ABB RobotStudio station: Projekt.rspag

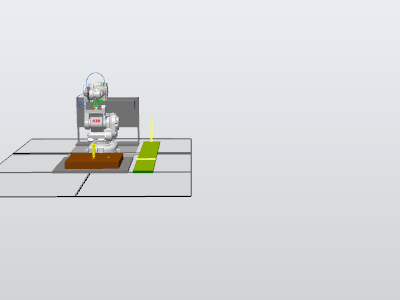
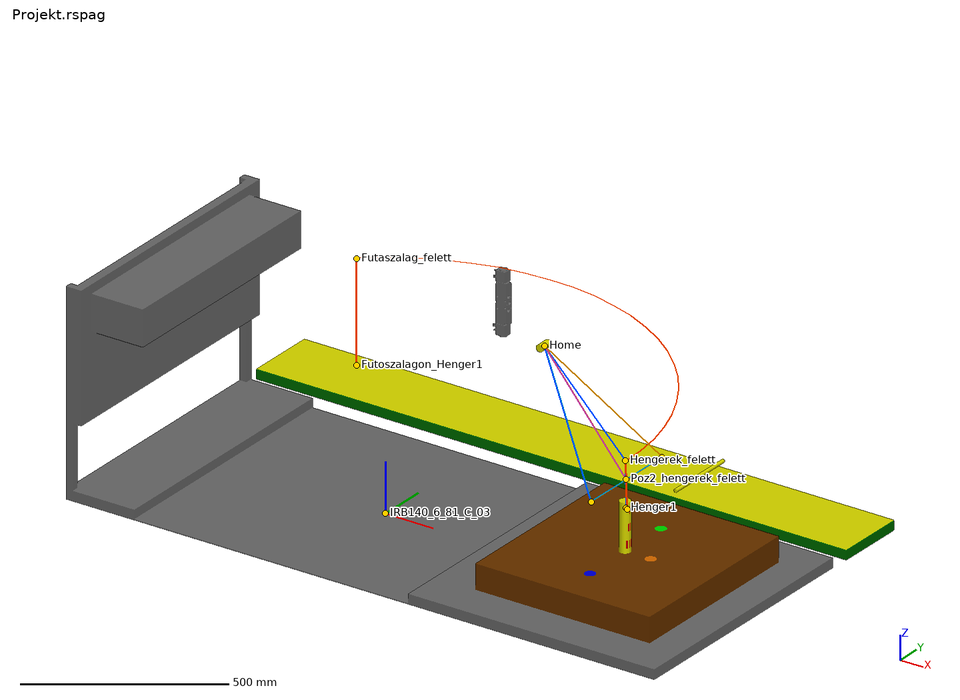
[picture v1: parts stored in the station drawn from their meshes, with robot base, taught points and paths (robot models come from the ABB library and are not in the file)]
--- station ---
Station hanoi_2022_RW6 (saved by RobotStudio 25.1.11167.1)
Controller IRB140_6_81
  mechanical unit ROB_1: IRB140_6_81_C_03, 6 joints, base frame (0, 0, 0) mm
Layout (positions relative to the parent item):
  - Henger1 [part] at (700, 0, 186) mm, rotated rx 0 ry 0 rz 180 deg, size 30.5 x 29.9 x 45 mm
  - Poz1 [part] at (700, 150, 96) mm, size 30 x 29.8 x 0 mm
  - Poz3 [part] at (700, 0, 96) mm, size 30 x 29.8 x 0 mm
  - SmatMefogo [smart component] at (450, 0, 647) mm, rotated rx -180 ry 0 rz -179.16 deg
      signals: DI Megfog, DI Elenged
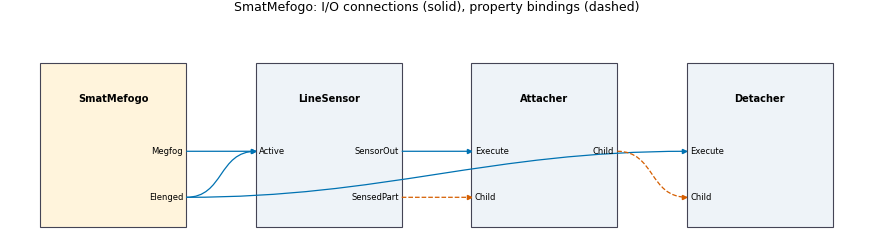
      connections:
        SmatMefogo.Megfog -> LineSensor.Active
        LineSensor.SensorOut -> Attacher.Execute
        SmatMefogo.Elenged -> LineSensor.Active
        SmatMefogo.Elenged -> Detacher.Execute
        LineSensor.SensedPart => Attacher.Child
        Attacher.Child => Detacher.Child
    - Megfogo [mechanism, from Libraries\Megfogo.rslib] at (0, 0, 0) mm, rotated rx 0 ry 0 rz -90 deg; joint values [0] (rad or m)
    - MegfogoTool [mechanism] at (0, 0, 0) mm
        TCP MyNewTool at (-15, 0, 70) mm, rotated rx -90 ry 0 rz -90 deg
        links: Dummy
    - LineSensor [smart component, from Components\LineSensor.rslib]
        properties: Start=[-0.0125 0.018 0.07]; End=[-0.0125 -0.019 0.07]; Radius=0.01; SensedPart=Henger1; SensedPoint=[0.704940063476562 -0.133748397827148 0.231000228881836]; Length=0.037; Tag=(none); SenseMultiple=false
      - _sensorPart_ [part], size 20 x 37 x 20 mm
    - Attacher [smart component, from Components\Attacher.rslib]
        properties: Parent=Megfogo; Flange=0; Child=Henger1; Mount=false; Offset=[0 0 0]; Orientation=[0 0 0]
    - Detacher [smart component, from Components\Detacher.rslib]
        properties: Child=Henger1; KeepPosition=true
  - SmartFSzalag [smart component] at (24.45, 0, 0) mm
      signals: DI Activate, DO SzalagErzekel
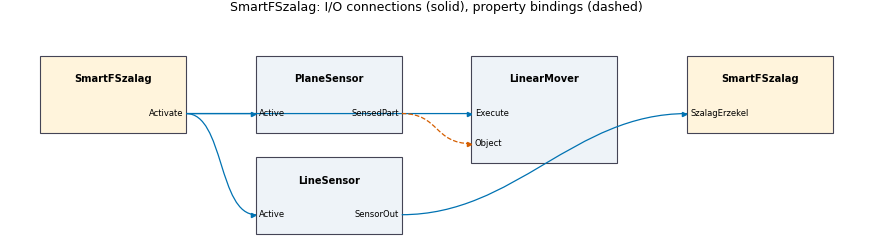
      connections:
        SmartFSzalag.Activate -> LinearMover.Execute
        SmartFSzalag.Activate -> PlaneSensor.Active
        SmartFSzalag.Activate -> LineSensor.Active
        LineSensor.SensorOut -> SmartFSzalag.SzalagErzekel
        PlaneSensor.SensedPart => LinearMover.Object
    - LinearMover [smart component, from Components\LinearMover.rslib]
        properties: Object=(none); Direction=[1 0 0]; Speed=0.1; Reference=Global; ReferenceObject=(none)
    - PlaneSensor [smart component, from Components\PlaneSensor.rslib]
        properties: Origin=[-0.7 0.425 0.027]; Axis1=[1.725 0 0]; Axis2=[0 0.2 0]; SensedPart=(none); Tag=(none); SenseMultiple=false
      - _sensorPart_ [part], size 1725 x 200 x 0 mm
    - FutoSzalag [part] at (-700, 425, 0) mm, size 1725 x 200 x 25 mm
    - LineSensor [smart component, from Components\LineSensor.rslib]
        properties: Start=[0.525 0.625 0.045]; End=[0.525 0.425 0.045]; Radius=0.005; SensedPart=(none); SensedPoint=[0 0 0]; Length=0.2; Tag=(none); SenseMultiple=false
      - _sensorPart_ [part], size 10 x 200 x 10 mm
  - Poz2 [part] at (-100, -100, 71) mm, size 30 x 29.8 x 0 mm
  - Asztal [part], size 1720 x 745 x 567 mm
  - Henger2 [part] at (700, 0, 141) mm, rotated rx 0 ry 0 rz 180 deg, size 30.5 x 29.9 x 45 mm
  - Henger3 [part] at (700, 0, 96) mm, rotated rx 0 ry 0 rz 180 deg, size 30.5 x 29.9 x 45 mm
  - Doboz [part] at (444.29, -260.35, 25.4) mm, size 510 x 540 x 70 mm
  - SolenoidValve [graphiccomponentgroup] at (400, -90, 651.5) mm, rotated rx 90 ry 0 rz 180 deg
    - coil_1 [part] at (16.04, 126.65, 10.8) mm, rotated rx 180 ry 0 rz -90 deg, size 29.6 x 38.6 x 22.3 mm
    - coil_2 [part] at (16, -15.19, 10.52) mm, rotated rx 0 ry 0 rz 90 deg, size 29.6 x 38.6 x 22.3 mm
    - solenoid [part], size 34 x 181.3 x 25.5 mm
  - IRB140_6_81_C_03 [mechanism, from %ABB.RobotStudio.Models.IRB140%\IRB140_6_81_C_G_03.rslib] at (0, 0, 0) mm; joint values [0, 0, 0, 0, 1.5708, -0.0146] (rad or m)
  - Poz4 [part] at (775, 0, 96) mm, size 30 x 29.8 x 0 mm
  - PneumaticsCable_1 [physicscable]
  - PneumaticsCable_2 [physicscable]
  - PneumaticsCable_3 [physicscable]
  - PneumaticsCable_4 [physicscable]
  - PneumaticsCable_5 [physicscable]
Attachment: SmatMefogo is attached to IRB140_6_81_C_03 / Link6
Attachment: SolenoidValve is attached to IRB140_6_81_C_03 / Link4
EventTableEntry 959: Group=, Trigger=DO10_1 960, Actions=[EventTableActionMechanicalPose 961], Comment=, ActivationMode=2, Cyclic=false
EventTableTriggerIO 960: IOValue=[1], IRC5Controller=? -1, Operator=0, SignalSource=IRB140_6_81 1488
EventTableActionMechanicalPose 961: VirtualSignal=, Mechanism=Megfogo 970, ToPoseName=Elenged, VirtualSignalValue=[1]
EventTableEntry 988: Group=, Trigger=DO10_2 989, Actions=[EventTableActionMechanicalPose 990], Comment=, ActivationMode=2, Cyclic=false
EventTableTriggerIO 989: IOValue=[1], IRC5Controller=? -1, Operator=0, SignalSource=IRB140_6_81 1488
EventTableActionMechanicalPose 990: VirtualSignal=, Mechanism=Megfogo 970, ToPoseName=Megfog, VirtualSignalValue=[1]
Collision set Critical_collision_1: Doboz, Asztal, FutoSzalag against Henger1, Henger2, Henger3, near miss 0.005 m
Collision set Critical_collision_2: SolenoidValve against Megfogo, near miss 0.01 m
Collision set Mandatory_collision_1: Megfogo against Henger1, Henger2, Henger3, near miss 0 m
Collision set Critical_collision_3: Megfogo against FutoSzalag, Asztal, Doboz, near miss 0.002 m
EventTableTriggerIO 2984: IOValue=[1], IRC5Controller=? -1, Operator=0, SignalSource=? -1
EventTableTriggerIO 2985: IOValue=[1], IRC5Controller=? -1, Operator=0, SignalSource=? -1
EventTableTriggerIO 3288: IOValue=[1], IRC5Controller=? -1, Operator=0, SignalSource=? -1
EventTableTriggerIO 3289: IOValue=[1], IRC5Controller=? -1, Operator=0, SignalSource=? -1
EventTableTriggerIO 3392: IOValue=[1], IRC5Controller=? -1, Operator=0, SignalSource=? -1
EventTableTriggerIO 3393: IOValue=[1], IRC5Controller=? -1, Operator=0, SignalSource=? -1
EventTableTriggerIO 3516: IOValue=[1], IRC5Controller=? -1, Operator=0, SignalSource=? -1
EventTableTriggerIO 3517: IOValue=[1], IRC5Controller=? -1, Operator=0, SignalSource=? -1
EventTableTriggerIO 4419: IOValue=[1], IRC5Controller=? -1, Operator=0, SignalSource=? -1
EventTableTriggerIO 4420: IOValue=[1], IRC5Controller=? -1, Operator=0, SignalSource=? -1
EventTableTriggerIO 4467: IOValue=[1], IRC5Controller=? -1, Operator=0, SignalSource=? -1
EventTableTriggerIO 4468: IOValue=[1], IRC5Controller=? -1, Operator=0, SignalSource=? -1
EventTableTriggerIO 4469: IOValue=[1], IRC5Controller=? -1, Operator=0, SignalSource=? -1
EventTableTriggerIO 4470: IOValue=[1], IRC5Controller=? -1, Operator=0, SignalSource=? -1
EventTableTriggerIO 4471: IOValue=[1], IRC5Controller=? -1, Operator=0, SignalSource=? -1
EventTableTriggerIO 4472: IOValue=[1], IRC5Controller=? -1, Operator=0, SignalSource=? -1
EventTableTriggerIO 4473: IOValue=[1], IRC5Controller=? -1, Operator=0, SignalSource=? -1
EventTableTriggerIO 4474: IOValue=[1], IRC5Controller=? -1, Operator=0, SignalSource=? -1
EventTableTriggerIO 4475: IOValue=[1], IRC5Controller=? -1, Operator=0, SignalSource=? -1
EventTableTriggerIO 4476: IOValue=[1], IRC5Controller=? -1, Operator=0, SignalSource=? -1
EventTableTriggerIO 4477: IOValue=[1], IRC5Controller=? -1, Operator=0, SignalSource=? -1
EventTableTriggerIO 4478: IOValue=[1], IRC5Controller=? -1, Operator=0, SignalSource=? -1
EventTableTriggerIO 4479: IOValue=[1], IRC5Controller=? -1, Operator=0, SignalSource=? -1
EventTableTriggerIO 4480: IOValue=[1], IRC5Controller=? -1, Operator=0, SignalSource=? -1
EventTableTriggerIO 4495: IOValue=[1], IRC5Controller=? -1, Operator=0, SignalSource=? -1
EventTableTriggerIO 4496: IOValue=[1], IRC5Controller=? -1, Operator=0, SignalSource=? -1
EventTableTriggerIO 5022: IOValue=[1], IRC5Controller=? -1, Operator=0, SignalSource=? -1
EventTableTriggerIO 5023: IOValue=[1], IRC5Controller=? -1, Operator=0, SignalSource=? -1
EventTableTriggerIO 5052: IOValue=[1], IRC5Controller=? -1, Operator=0, SignalSource=? -1
EventTableTriggerIO 5053: IOValue=[1], IRC5Controller=? -1, Operator=0, SignalSource=? -1
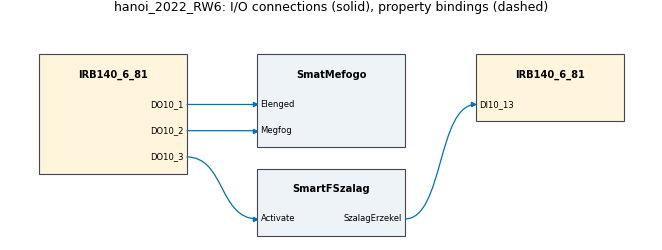
Station logic (signal -> signal, property => property):
  IRB140_6_81.DO10_1 -> SmatMefogo.Elenged
  IRB140_6_81.DO10_2 -> SmatMefogo.Megfog
  IRB140_6_81.DO10_3 -> SmartFSzalag.Activate
  SmartFSzalag.SzalagErzekel -> IRB140_6_81.DI10_13
Targets, tools, work objects and paths stored in the station and not in the controller backup, written as RAPID:
! task T_ROB1
MODULE CalibData
  PERS tooldata MegfogoTool:=[TRUE,[[-15,0,70],[0.5,-0.5,0.5,-0.5]],[1,[0,0,1],[1,0,0,0],0,0,0]];
ENDMODULE

! task T_ROB1
MODULE Module1
  CONST robtarget Poz3_:=[[706.158574635,-148.692803379,203.565715779],[0.488723977,0.511027269,-0.511027275,-0.488723979],[-1,0,-1,0],[9E+09,9E+09,9E+09,9E+09,9E+09,9E+09]];
ENDMODULE


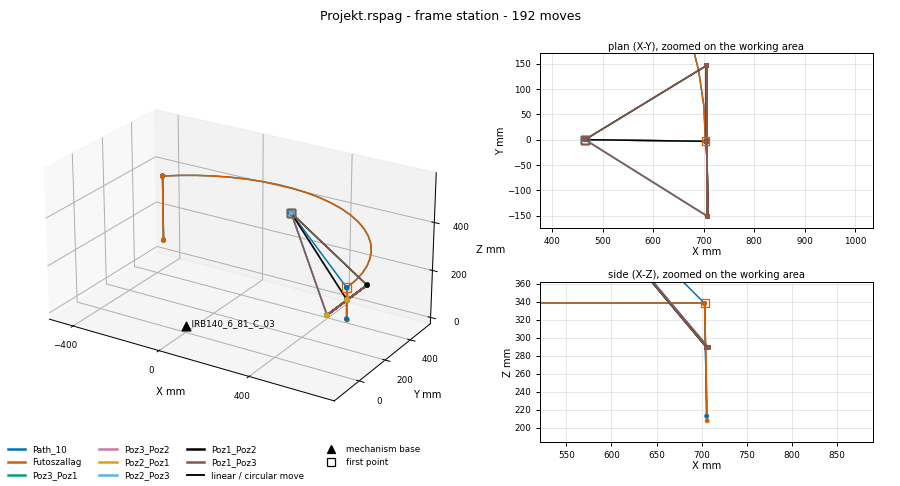
[picture p0: tool path of Projekt.rspag in frame station, 192 of 276 moves have a stored position in this frame; points joined in program order, loops and branches not executed]
--- Backups/IRB140_6_81/RAPID/TASK1/PROGMOD/CalibData.mod ---
MODULE CalibData
    PERS tooldata MyNewTool:=[TRUE,[[-15,0,70],[0.5,-0.5,0.5,-0.5]],[1,[0,0,1],[1,0,0,0],0,0,0]];
ENDMODULE

--- Backups/IRB140_6_81/RAPID/TASK1/PROGMOD/Module1.mod ---
MODULE Module1

    !-----------------------------
    ! Céltárgyak (robtarget-ek)
    !-----------------------------

    CONST robtarget Home:=[[464.998399046,0.219148469,577],[0.50363923,0.50363923,-0.496334087,-0.496334087],[0,0,-1,0],[9E+09,9E+09,9E+09,9E+09,9E+09,9E+09]];
    CONST robtarget Target_10:=[[465.000006606,0,511.354787728],[0.500000003,0.499999997,-0.499999997,-0.500000003],[0,0,0,0],[9E+09,9E+09,9E+09,9E+09,9E+09,9E+09]];
    CONST robtarget Target_20:=[[464.999999789,63.315024893,511.354787009],[0.500000017,0.499999983,-0.499999987,-0.500000013],[0,0,0,0],[9E+09,9E+09,9E+09,9E+09,9E+09,9E+09]];
    CONST robtarget Target_30:=[[465.000004629,63.315025575,573.930963746],[0.500000008,0.499999992,-0.499999994,-0.500000006],[0,0,0,0],[9E+09,9E+09,9E+09,9E+09,9E+09,9E+09]];
    CONST robtarget K:=[[465.000011429,-20.081921365,542.489098176],[0.49999989,0.500000109,-0.500000111,-0.49999989],[-1,0,-1,0],[9E+09,9E+09,9E+09,9E+09,9E+09,9E+09]];
    CONST robtarget Henger2_felett:=[[703.330980263,-3.101798952,338.097192514],[0.500000018,0.499999982,-0.499999982,-0.500000018],[-1,0,-1,0],[9E+09,9E+09,9E+09,9E+09,9E+09,9E+09]];
    CONST robtarget Henger2:=[[703.330979486,-3.101798949,122.952378135],[0.500000003,0.499999997,-0.499999997,-0.500000003],[-1,0,-1,0],[9E+09,9E+09,9E+09,9E+09,9E+09,9E+09]];
    CONST robtarget Koriv_pont:=[[468.348006502,524.723006699,338.097192514],[0.661244366,0.661244318,-0.250511308,-0.250511327],[0,-1,-1,0],[9E+09,9E+09,9E+09,9E+09,9E+09,9E+09]];
    CONST robtarget Futaszalag_felett:=[[-458.230855192,533.580815511,338.096713631],[0.662525774,0.662525349,0.247102897,0.247103054],[1,-1,-1,0],[9E+09,9E+09,9E+09,9E+09,9E+09,9E+09]];
    CONST robtarget Futoszalag_vege:=[[-458.230834781,533.580796254,152.170174534],[0.662525692,0.662525413,0.247102906,0.247103092],[1,-1,-1,0],[9E+09,9E+09,9E+09,9E+09,9E+09,9E+09]];
    CONST robtarget Hengerek_felett:=[[703.330980263,-3.101798952,338.097192514],[0.500000018,0.499999982,-0.499999982,-0.500000018],[-1,0,-1,0],[9E+09,9E+09,9E+09,9E+09,9E+09,9E+09]];
    CONST robtarget Henger1:=[[705.540590209,-3.101798785,213.051995114],[0.500000003,0.499999997,-0.499999997,-0.500000003],[-1,0,-1,0],[9E+09,9E+09,9E+09,9E+09,9E+09,9E+09]];
    CONST robtarget Futoszalag_felett1:=[[-458.230781636,533.580759154,27.200885596],[0.662525692,0.662525413,0.247102906,0.247103092],[1,-1,-1,0],[9E+09,9E+09,9E+09,9E+09,9E+09,9E+09]];
    CONST robtarget Futoszalagon_Henger1:=[[-458.230849578,533.580833502,53.435741124],[0.662525708,0.66252543,0.247102862,0.247103049],[1,-1,-1,0],[9E+09,9E+09,9E+09,9E+09,9E+09,9E+09]];
    CONST robtarget Poz3_hengerek_felett:=[[707.440014419,-151.570005718,289.3],[0.499999997,0.500000003,-0.500000005,-0.499999995],[-1,0,-1,0],[9E+09,9E+09,9E+09,9E+09,9E+09,9E+09]];
    CONST robtarget Poz2_hengerek_felett:=[[705.540594643,-3.101798805,289.3],[0.499999996,0.500000004,-0.500000004,-0.499999996],[-1,0,-1,0],[9E+09,9E+09,9E+09,9E+09,9E+09,9E+09]];
    CONST robtarget Poz1_hengerek_felett:=[[705.539993286,146.89999968,289.3],[0.499999995,0.500000005,-0.500000003,-0.499999997],[0,0,0,0],[9E+09,9E+09,9E+09,9E+09,9E+09,9E+09]];
    CONST robtarget Poz1_also:=[[706.158568656,148.13220538,120.859568206],[0.488723989,0.511027265,-0.511027263,-0.488723984],[0,-1,0,0],[9E+09,9E+09,9E+09,9E+09,9E+09,9E+09]];
    CONST robtarget Poz1_felso:=[[706.158581923,150.789795781,200.699837478],[0.488723963,0.511027284,-0.51102728,-0.488723973],[0,-1,0,0],[9E+09,9E+09,9E+09,9E+09,9E+09,9E+09]];
    CONST robtarget Poz1_kozepso:=[[706.158576433,149.655297873,161.602721107],[0.488723973,0.511027276,-0.511027274,-0.488723978],[0,-1,0,0],[9E+09,9E+09,9E+09,9E+09,9E+09,9E+09]];
    CONST robtarget Poz2_also:=[[706.158557063,0.931775994,120.859559008],[0.488724,0.511027251,-0.511027251,-0.488724],[0,-1,0,0],[9E+09,9E+09,9E+09,9E+09,9E+09,9E+09]];
    CONST robtarget Poz2_felso:=[[706.158575812,0.212934892,207.997391033],[0.48872398,0.511027271,-0.511027271,-0.48872398],[0,-1,0,0],[9E+09,9E+09,9E+09,9E+09,9E+09,9E+09]];
    CONST robtarget Poz2_kozepso:=[[706.158568247,0.212934889,161.602696818],[0.488723988,0.511027263,-0.511027263,-0.488723988],[0,-1,0,0],[9E+09,9E+09,9E+09,9E+09,9E+09,9E+09]];
    CONST robtarget Poz3_also:=[[706.158576885,-147.845803893,120.859626189],[0.488723975,0.511027273,-0.511027279,-0.488723974],[-1,0,-1,0],[9E+09,9E+09,9E+09,9E+09,9E+09,9E+09]];
    CONST robtarget Poz3_felso:=[[706.158578379,-148.69280434,205.909014134],[0.48872397,0.511027274,-0.511027286,-0.48872397],[-1,0,-1,0],[9E+09,9E+09,9E+09,9E+09,9E+09,9E+09]];
    CONST robtarget Poz3_kozepso:=[[706.158568337,-148.692802057,161.602704679],[0.488723987,0.511027264,-0.511027263,-0.488723988],[-1,0,-1,0],[9E+09,9E+09,9E+09,9E+09,9E+09,9E+09]];

    !-----------------------------
    ! Digitális kimenetek használata
    !-----------------------------
    PROC Megfog()
    ! Megfogó zárása
        PulseDO DO10_2;
        WaitTime 1;
    ENDPROC

    PROC Elenged()
        PulseDO DO10_1;   ! Megfogó nyitása
        WaitTime 1;
    ENDPROC


    PROC FutoszalagIndit()
        SetDO DO10_3, 1;
        WaitTime 1;
    ENDPROC

    PROC FutoszalagStop()
        SetDO DO10_3, 0;
        WaitTime 1;
    ENDPROC

    !-----------------------------
    ! Fo program - 1. mérföldko
    !-----------------------------

PROC main()
    VAR num valasz := -1;
    VAR num start_poz := -1;
    VAR num cel_poz := -1;

    TPReadFK valasz, "Elindítod a szimulációt?", "Igen", "Nem", "", "", "";
    IF valasz = 2 THEN
        TPWrite("A szimuláció megszakítva.");
        RETURN;
    ENDIF

    TPReadFK start_poz, "Hol vannak most a hengerek?", "Poz1", "Poz2", "Poz3", "", "";

    IF start_poz = 1 THEN
        TPReadFK cel_poz, "Hova rakjuk a hengereket?", "Poz2", "Poz3", "", "", "";
        IF cel_poz = 1 THEN
            Poz1_poz2;
            RETURN;
        ELSEIF cel_poz = 2 THEN
            Poz1_poz3;
            RETURN;
        ENDIF

    ELSEIF start_poz = 2 THEN
        TPReadFK cel_poz, "Hova rakjuk a hengereket?", "Poz1", "Poz3", "", "", "";
        IF cel_poz = 1 THEN
            Poz2_poz1;
            RETURN;
        ELSEIF cel_poz = 2 THEN
            Poz2_poz3;
            RETURN;
        ENDIF

    ELSEIF start_poz = 3 THEN
        TPReadFK cel_poz, "Hova rakjuk a hengereket?", "Poz1", "Poz2", "", "", "";
        IF cel_poz = 1 THEN
            Poz3_poz1;
            RETURN;
        ELSEIF cel_poz = 2 THEN
            Poz3_poz2;
            RETURN;
        ENDIF

    ELSE
        TPWrite("Érvénytelen kezdopozíció!");
        RETURN;
    ENDIF
ENDPROC


    PROC Path_10()
        MoveL Home,v400,fine,MyNewTool\WObj:=wobj0;
        MoveL Hengerek_felett,v400,fine,MyNewTool\WObj:=wobj0;
        MoveL Henger1,v100,fine,MyNewTool\WObj:=wobj0;
        Megfog;
        MoveL Hengerek_felett,v400,fine,MyNewTool\WObj:=wobj0;
        MoveC Koriv_pont,Futaszalag_felett,v400,fine,MyNewTool\WObj:=wobj0;
        MoveL Futoszalagon_Henger1,v100,fine,MyNewTool\WObj:=wobj0;
        Elenged;
        MoveL Futaszalag_felett,v100,fine,MyNewTool\WObj:=wobj0;
        FutoszalagIndit;
        WaitDI DI10_13, 1;
        FutoszalagStop;
    ENDPROC
    PROC Futoszallag()
        MoveL Hengerek_felett,v400,fine,MyNewTool\WObj:=wobj0;
        MoveL Poz2_felso,v100,fine,MyNewTool\WObj:=wobj0;
        Megfog;
        MoveL Hengerek_felett,v400,fine,MyNewTool\WObj:=wobj0;
        MoveC Koriv_pont,Futaszalag_felett,v400,fine,MyNewTool\WObj:=wobj0;
        MoveL Futoszalagon_Henger1,v100,fine,MyNewTool\WObj:=wobj0;
        Elenged;
        MoveL Futaszalag_felett,v100,fine,MyNewTool\WObj:=wobj0;
        FutoszalagIndit;
        WaitDI DI10_13,1;
        FutoszalagStop;
    ENDPROC

PROC Poz3_Poz1()
    CONST num hMag := 45;
    CONST num felOffset := hMag / 2;
    MoveL Home, v100, fine, MyNewTool;

    Elenged;

    ! 1. Poz3 felülrol 1. henger ? Poz1 alulra
    MoveL Poz3_hengerek_felett, v100, fine, MyNewTool;
    MoveL Offs(Poz3_hengerek_felett, 0, 0, -80.8 + felOffset), v100, fine, MyNewTool;  ! felül
    Megfog;
    MoveL Poz3_hengerek_felett, v100, fine, MyNewTool;
    MoveL Poz1_hengerek_felett, v100, fine, MyNewTool;
    MoveL Offs(Poz1_hengerek_felett, 0, 0, -170.8 + felOffset), v100, fine, MyNewTool; ! alul
    Elenged;
    MoveL Poz1_hengerek_felett, v100, fine, MyNewTool;

    ! 2. Poz3 középso 2. henger ? Poz2 alulra
    MoveL Poz3_hengerek_felett, v100, fine, MyNewTool;
    MoveL Offs(Poz3_hengerek_felett, 0, 0, -125.8 + felOffset), v100, fine, MyNewTool; ! középso
    Megfog;
    MoveL Poz3_hengerek_felett, v100, fine, MyNewTool;
    MoveL Poz2_hengerek_felett, v100, fine, MyNewTool;
    MoveL Offs(Poz2_hengerek_felett, 0, 0, -170.8 + felOffset), v100, fine, MyNewTool; ! alul
    Elenged;
    MoveL Poz2_hengerek_felett, v100, fine, MyNewTool;

    ! 3. Poz1 alsóról 1. henger ? Poz2 középre
    MoveL Poz1_hengerek_felett, v100, fine, MyNewTool;
    MoveL Offs(Poz1_hengerek_felett, 0, 0, -170.8 + felOffset), v100, fine, MyNewTool; ! alul
    Megfog;
    MoveL Poz1_hengerek_felett, v100, fine, MyNewTool;
    MoveL Poz2_hengerek_felett, v100, fine, MyNewTool;
    MoveL Offs(Poz2_hengerek_felett, 0, 0, -125.8 + felOffset), v100, fine, MyNewTool; ! középso
    Elenged;
    MoveL Poz2_hengerek_felett, v100, fine, MyNewTool;

    ! 4. Poz3 alsóról 3. henger ? Poz1 alsóra
    MoveL Poz3_hengerek_felett, v100, fine, MyNewTool;
    MoveL Offs(Poz3_hengerek_felett, 0, 0, -170.8 + felOffset), v100, fine, MyNewTool; ! alul
    Megfog;
    MoveL Poz3_hengerek_felett, v100, fine, MyNewTool;
    MoveL Poz1_hengerek_felett, v100, fine, MyNewTool;
    MoveL Offs(Poz1_hengerek_felett, 0, 0, -170.8 + felOffset), v100, fine, MyNewTool; ! alul
    Elenged;
    MoveL Poz1_hengerek_felett, v100, fine, MyNewTool;

    ! 5. Poz2 középsorol 1. henger ? Poz3 alsóra
    MoveL Poz2_hengerek_felett, v100, fine, MyNewTool;
    MoveL Offs(Poz2_hengerek_felett, 0, 0, -125.8 + felOffset), v100, fine, MyNewTool; ! középso
    Megfog;
    MoveL Poz2_hengerek_felett, v100, fine, MyNewTool;
    MoveL Poz3_hengerek_felett, v100, fine, MyNewTool;
    MoveL Offs(Poz3_hengerek_felett, 0, 0, -170.8 + felOffset), v100, fine, MyNewTool; ! alul
    Elenged;
    MoveL Poz3_hengerek_felett, v100, fine, MyNewTool;

    ! 6. Poz2 alsóról 2. henger ? Poz1 középre
    MoveL Poz2_hengerek_felett, v100, fine, MyNewTool;
    MoveL Offs(Poz2_hengerek_felett, 0, 0, -170.8 + felOffset), v100, fine, MyNewTool; ! alul
    Megfog;
    MoveL Poz2_hengerek_felett, v100, fine, MyNewTool;
    MoveL Poz1_hengerek_felett, v100, fine, MyNewTool;
    MoveL Offs(Poz1_hengerek_felett, 0, 0, -125.8 + felOffset), v100, fine, MyNewTool; ! középso
    Elenged;
    MoveL Poz1_hengerek_felett, v100, fine, MyNewTool;

    ! 7. Poz3 alsóról 1. henger ? Poz1 felülre
    MoveL Poz3_hengerek_felett, v100, fine, MyNewTool;
    MoveL Offs(Poz3_hengerek_felett, 0, 0, -170.8 + felOffset), v100, fine, MyNewTool; ! alul
    Megfog;
    MoveL Poz3_hengerek_felett, v100, fine, MyNewTool;
    MoveL Poz1_hengerek_felett, v100, fine, MyNewTool;
    MoveL Offs(Poz1_hengerek_felett, 0, 0, -80.8 + felOffset), v100, fine, MyNewTool; ! felül
    Elenged;
    MoveL Poz1_hengerek_felett, v100, fine, MyNewTool;

    MoveL Home, v100, fine, MyNewTool;
ENDPROC

PROC Poz3_Poz2()
CONST num hMag := 45;
CONST num felOffset := hMag / 2;

MoveL Home, v100, fine, MyNewTool\WObj:=wobj0;

! 1. Poz3 felülrol (1. henger) ? Poz2 alulra
MoveL Poz3_hengerek_felett, v100, fine, MyNewTool;
MoveL Offs(Poz3_hengerek_felett, 0, 0, -80.8 + felOffset), v100, fine, MyNewTool;
Megfog;
MoveL Poz3_hengerek_felett, v100, fine, MyNewTool;
MoveL Poz2_hengerek_felett, v100, fine, MyNewTool;
MoveL Offs(Poz2_hengerek_felett, 0, 0, -170.8 + felOffset), v100, fine, MyNewTool;
Elenged;
MoveL Poz2_hengerek_felett, v100, fine, MyNewTool;

! 2. Poz3 középrol (2. henger) ? Poz1 alulra
MoveL Poz3_hengerek_felett, v100, fine, MyNewTool;
MoveL Offs(Poz3_hengerek_felett, 0, 0, -125.8 + felOffset), v100, fine, MyNewTool;
Megfog;
MoveL Poz3_hengerek_felett, v100, fine, MyNewTool;
MoveL Poz1_hengerek_felett, v100, fine, MyNewTool;
MoveL Offs(Poz1_hengerek_felett, 0, 0, -170.8 + felOffset), v100, fine, MyNewTool;
Elenged;
MoveL Poz1_hengerek_felett, v100, fine, MyNewTool;

! 3. Poz2 alulról (1. henger) ? Poz1 középre
MoveL Poz2_hengerek_felett, v100, fine, MyNewTool;
MoveL Offs(Poz2_hengerek_felett, 0, 0, -170.8 + felOffset), v100, fine, MyNewTool;
Megfog;
MoveL Poz2_hengerek_felett, v100, fine, MyNewTool;
MoveL Poz1_hengerek_felett, v100, fine, MyNewTool;
MoveL Offs(Poz1_hengerek_felett, 0, 0, -125.8 + felOffset), v100, fine, MyNewTool;
Elenged;
MoveL Poz1_hengerek_felett, v100, fine, MyNewTool;

! 4. Poz3 alulról (3. henger) ? Poz2 alulra
MoveL Poz3_hengerek_felett, v100, fine, MyNewTool;
MoveL Offs(Poz3_hengerek_felett, 0, 0, -170.8 + felOffset), v100, fine, MyNewTool;
Megfog;
MoveL Poz3_hengerek_felett, v100, fine, MyNewTool;
MoveL Poz2_hengerek_felett, v100, fine, MyNewTool;
MoveL Offs(Poz2_hengerek_felett, 0, 0, -170.8 + felOffset), v100, fine, MyNewTool;
Elenged;
MoveL Poz2_hengerek_felett, v100, fine, MyNewTool;

! 5. Poz1 középrol (1. henger) ? Poz3 alulra
MoveL Poz1_hengerek_felett, v100, fine, MyNewTool;
MoveL Offs(Poz1_hengerek_felett, 0, 0, -125.8 + felOffset), v100, fine, MyNewTool;
Megfog;
MoveL Poz1_hengerek_felett, v100, fine, MyNewTool;
MoveL Poz3_hengerek_felett, v100, fine, MyNewTool;
MoveL Offs(Poz3_hengerek_felett, 0, 0, -170.8 + felOffset), v100, fine, MyNewTool;
Elenged;
MoveL Poz3_hengerek_felett, v100, fine, MyNewTool;

! 6. Poz1 alulról (2. henger) ? Poz2 középre
MoveL Poz1_hengerek_felett, v100, fine, MyNewTool;
MoveL Offs(Poz1_hengerek_felett, 0, 0, -170.8 + felOffset), v100, fine, MyNewTool;
Megfog;
MoveL Poz1_hengerek_felett, v100, fine, MyNewTool;
MoveL Poz2_hengerek_felett, v100, fine, MyNewTool;
MoveL Offs(Poz2_hengerek_felett, 0, 0, -125.8 + felOffset), v100, fine, MyNewTool;
Elenged;
MoveL Poz2_hengerek_felett, v100, fine, MyNewTool;

! 7. Poz3 alulról (1. henger) ? Poz2 felülre
MoveL Poz3_hengerek_felett, v100, fine, MyNewTool;
MoveL Offs(Poz3_hengerek_felett, 0, 0, -170.8 + felOffset), v100, fine, MyNewTool;
Megfog;
MoveL Poz3_hengerek_felett, v100, fine, MyNewTool;
MoveL Poz2_hengerek_felett, v100, fine, MyNewTool;
MoveL Offs(Poz2_hengerek_felett, 0, 0, -80.8 + felOffset), v100, fine, MyNewTool;
Elenged;
MoveL Poz2_hengerek_felett, v100, fine, MyNewTool;

MoveL Home, v100, fine, MyNewTool;

ENDPROC

PROC Poz2_Poz1()
    CONST num hMag := 45;             ! Henger magasság
    CONST num felOffset := hMag / 2;  ! Középre fogunk

    MoveL Home, v100, fine, MyNewTool\WObj:=wobj0;

    ! 1. Poz2 felülrol ? Poz1 alulra
    MoveL Poz2_hengerek_felett, v100, fine, MyNewTool\WObj:=wobj0;
    MoveL Offs(Poz2_hengerek_felett, 0, 0, -80.8 + felOffset), v100, fine, MyNewTool\WObj:=wobj0;
    Megfog;
    MoveL Poz2_hengerek_felett, v100, fine, MyNewTool\WObj:=wobj0;
    MoveL Poz1_hengerek_felett, v100, fine, MyNewTool\WObj:=wobj0;
    MoveL Offs(Poz1_hengerek_felett, 0, 0, -170.8 + felOffset), v100, fine, MyNewTool\WObj:=wobj0;
    Elenged;
    MoveL Poz1_hengerek_felett, v100, fine, MyNewTool\WObj:=wobj0;

    ! 2. Poz2 középrol ? Poz3 alulra
    MoveL Poz2_hengerek_felett, v100, fine, MyNewTool\WObj:=wobj0;
    MoveL Offs(Poz2_hengerek_felett, 0, 0, -125.8 + felOffset), v100, fine, MyNewTool\WObj:=wobj0;
    Megfog;
    MoveL Poz2_hengerek_felett, v100, fine, MyNewTool\WObj:=wobj0;
    MoveL Poz3_hengerek_felett, v100, fine, MyNewTool\WObj:=wobj0;
    MoveL Offs(Poz3_hengerek_felett, 0, 0, -170.8 + felOffset), v100, fine, MyNewTool\WObj:=wobj0;
    Elenged;
    MoveL Poz3_hengerek_felett, v100, fine, MyNewTool\WObj:=wobj0;

    ! 3. Poz1 alulról ? Poz3 középre
    MoveL Poz1_hengerek_felett, v100, fine, MyNewTool\WObj:=wobj0;
    MoveL Offs(Poz1_hengerek_felett, 0, 0, -170.8 + felOffset), v100, fine, MyNewTool\WObj:=wobj0;
    Megfog;
    MoveL Poz1_hengerek_felett, v100, fine, MyNewTool\WObj:=wobj0;
    MoveL Poz3_hengerek_felett, v100, fine, MyNewTool\WObj:=wobj0;
    MoveL Offs(Poz3_hengerek_felett, 0, 0, -125.8 + felOffset), v100, fine, MyNewTool\WObj:=wobj0;
    Elenged;
    MoveL Poz3_hengerek_felett, v100, fine, MyNewTool\WObj:=wobj0;

    ! 4. Poz2 alulról ? Poz1 alulra
    MoveL Poz2_hengerek_felett, v100, fine, MyNewTool\WObj:=wobj0;
    MoveL Offs(Poz2_hengerek_felett, 0, 0, -170.8 + felOffset), v100, fine, MyNewTool\WObj:=wobj0;
    Megfog;
    MoveL Poz2_hengerek_felett, v100, fine, MyNewTool\WObj:=wobj0;
    MoveL Poz1_hengerek_felett, v100, fine, MyNewTool\WObj:=wobj0;
    MoveL Offs(Poz1_hengerek_felett, 0, 0, -170.8 + felOffset), v100, fine, MyNewTool\WObj:=wobj0;
    Elenged;
    MoveL Poz1_hengerek_felett, v100, fine, MyNewTool\WObj:=wobj0;

    ! 5. Poz3 középrol ? Poz2 alulra
    MoveL Poz3_hengerek_felett, v100, fine, MyNewTool\WObj:=wobj0;
    MoveL Offs(Poz3_hengerek_felett, 0, 0, -125.8 + felOffset), v100, fine, MyNewTool\WObj:=wobj0;
    Megfog;
    MoveL Poz3_hengerek_felett, v100, fine, MyNewTool\WObj:=wobj0;
    MoveL Poz2_hengerek_felett, v100, fine, MyNewTool\WObj:=wobj0;
    MoveL Offs(Poz2_hengerek_felett, 0, 0, -170.8 + felOffset), v100, fine, MyNewTool\WObj:=wobj0;
    Elenged;
    MoveL Poz2_hengerek_felett, v100, fine, MyNewTool\WObj:=wobj0;

    ! 6. Poz3 alulról ? Poz1 középre
    MoveL Poz3_hengerek_felett, v100, fine, MyNewTool\WObj:=wobj0;
    MoveL Offs(Poz3_hengerek_felett, 0, 0, -170.8 + felOffset), v100, fine, MyNewTool\WObj:=wobj0;
    Megfog;
    MoveL Poz3_hengerek_felett, v100, fine, MyNewTool\WObj:=wobj0;
    MoveL Poz1_hengerek_felett, v100, fine, MyNewTool\WObj:=wobj0;
    MoveL Offs(Poz1_hengerek_felett, 0, 0, -125.8 + felOffset), v100, fine, MyNewTool\WObj:=wobj0;
    Elenged;
    MoveL Poz1_hengerek_felett, v100, fine, MyNewTool\WObj:=wobj0;

    ! 7. Poz2 alulról ? Poz1 felülre
    MoveL Poz2_hengerek_felett, v100, fine, MyNewTool\WObj:=wobj0;
    MoveL Offs(Poz2_hengerek_felett, 0, 0, -170.8 + felOffset), v100, fine, MyNewTool\WObj:=wobj0;
    Megfog;
    MoveL Poz2_hengerek_felett, v100, fine, MyNewTool\WObj:=wobj0;
    MoveL Poz1_hengerek_felett, v100, fine, MyNewTool\WObj:=wobj0;
    MoveL Offs(Poz1_hengerek_felett, 0, 0, -80.8 + felOffset), v100, fine, MyNewTool\WObj:=wobj0;
    Elenged;
    MoveL Poz1_hengerek_felett, v100, fine, MyNewTool\WObj:=wobj0;
ENDPROC

PROC Poz2_Poz3()
    CONST num hMag := 45;
    CONST num felOffset := hMag / 2;

    MoveL Home, v100, fine, MyNewTool\WObj:=wobj0;

    ! 1. Poz2 felülrol (1. henger) ? Poz3 alulra
    MoveL Poz2_hengerek_felett, v100, fine, MyNewTool;
    MoveL Offs(Poz2_hengerek_felett, 0, 0, -80.8 + felOffset), v100, fine, MyNewTool;
    Megfog;
    MoveL Poz2_hengerek_felett, v100, fine, MyNewTool;
    MoveL Poz3_hengerek_felett, v100, fine, MyNewTool;
    MoveL Offs(Poz3_hengerek_felett, 0, 0, -170.8 + felOffset), v100, fine, MyNewTool;
    Elenged;
    MoveL Poz3_hengerek_felett, v100, fine, MyNewTool;

    ! 2. Poz2 középrol (2. henger) ? Poz1 alulra
    MoveL Poz2_hengerek_felett, v100, fine, MyNewTool;
    MoveL Offs(Poz2_hengerek_felett, 0, 0, -125.8 + felOffset), v100, fine, MyNewTool;
    Megfog;
    MoveL Poz2_hengerek_felett, v100, fine, MyNewTool;
    MoveL Poz1_hengerek_felett, v100, fine, MyNewTool;
    MoveL Offs(Poz1_hengerek_felett, 0, 0, -170.8 + felOffset), v100, fine, MyNewTool;
    Elenged;
    MoveL Poz1_hengerek_felett, v100, fine, MyNewTool;

    ! 3. Poz3 alulról (1. henger) ? Poz1 középre
    MoveL Poz3_hengerek_felett, v100, fine, MyNewTool;
    MoveL Offs(Poz3_hengerek_felett, 0, 0, -170.8 + felOffset), v100, fine, MyNewTool;
    Megfog;
    MoveL Poz3_hengerek_felett, v100, fine, MyNewTool;
    MoveL Poz1_hengerek_felett, v100, fine, MyNewTool;
    MoveL Offs(Poz1_hengerek_felett, 0, 0, -125.8 + felOffset), v100, fine, MyNewTool;
    Elenged;
    MoveL Poz1_hengerek_felett, v100, fine, MyNewTool;

    ! 4. Poz2 alulról (3. henger) ? Poz3 alulra
    MoveL Poz2_hengerek_felett, v100, fine, MyNewTool;
    MoveL Offs(Poz2_hengerek_felett, 0, 0, -170.8 + felOffset), v100, fine, MyNewTool;
    Megfog;
    MoveL Poz2_hengerek_felett, v100, fine, MyNewTool;
    MoveL Poz3_hengerek_felett, v100, fine, MyNewTool;
    MoveL Offs(Poz3_hengerek_felett, 0, 0, -170.8 + felOffset), v100, fine, MyNewTool;
    Elenged;
    MoveL Poz3_hengerek_felett, v100, fine, MyNewTool;

    ! 5. Poz1 középrol (1. henger) ? Poz2 alulra
    MoveL Poz1_hengerek_felett, v100, fine, MyNewTool;
    MoveL Offs(Poz1_hengerek_felett, 0, 0, -125.8 + felOffset), v100, fine, MyNewTool;
    Megfog;
    MoveL Poz1_hengerek_felett, v100, fine, MyNewTool;
    MoveL Poz2_hengerek_felett, v100, fine, MyNewTool;
    MoveL Offs(Poz2_hengerek_felett, 0, 0, -170.8 + felOffset), v100, fine, MyNewTool;
    Elenged;
    MoveL Poz2_hengerek_felett, v100, fine, MyNewTool;

    ! 6. Poz1 alulról (2. henger) ? Poz3 középre
    MoveL Poz1_hengerek_felett, v100, fine, MyNewTool;
    MoveL Offs(Poz1_hengerek_felett, 0, 0, -170.8 + felOffset), v100, fine, MyNewTool;
    Megfog;
    MoveL Poz1_hengerek_felett, v100, fine, MyNewTool;
    MoveL Poz3_hengerek_felett, v100, fine, MyNewTool;
    MoveL Offs(Poz3_hengerek_felett, 0, 0, -125.8 + felOffset), v100, fine, MyNewTool;
    Elenged;
    MoveL Poz3_hengerek_felett, v100, fine, MyNewTool;

    ! 7. Poz2 alulról (1. henger) ? Poz3 felülre
    MoveL Poz2_hengerek_felett, v100, fine, MyNewTool;
    MoveL Offs(Poz2_hengerek_felett, 0, 0, -170.8 + felOffset), v100, fine, MyNewTool;
    Megfog;
    MoveL Poz2_hengerek_felett, v100, fine, MyNewTool;
    MoveL Poz3_hengerek_felett, v100, fine, MyNewTool;
    MoveL Offs(Poz3_hengerek_felett, 0, 0, -80.8 + felOffset), v100, fine, MyNewTool;
    Elenged;
    MoveL Poz3_hengerek_felett, v100, fine, MyNewTool;

    MoveL Home, v100, fine, MyNewTool;
ENDPROC

PROC Poz1_Poz2()
    CONST num hMag := 45;
    CONST num felOffset := hMag / 2;

    MoveL Home, v100, fine, MyNewTool\WObj:=wobj0;

    ! 1. Poz1 felülrol (1. henger) ? Poz2 alulra
    MoveL Poz1_hengerek_felett, v100, fine, MyNewTool;
    MoveL Offs(Poz1_hengerek_felett, 0, 0, -80.8 + felOffset), v100, fine, MyNewTool;
    Megfog;
    MoveL Poz1_hengerek_felett, v100, fine, MyNewTool;
    MoveL Poz2_hengerek_felett, v100, fine, MyNewTool;
    MoveL Offs(Poz2_hengerek_felett, 0, 0, -170.8 + felOffset), v100, fine, MyNewTool;
    Elenged;
    MoveL Poz2_hengerek_felett, v100, fine, MyNewTool;

    ! 2. Poz1 középrol (2. henger) ? Poz3 alulra
    MoveL Poz1_hengerek_felett, v100, fine, MyNewTool;
    MoveL Offs(Poz1_hengerek_felett, 0, 0, -125.8 + felOffset), v100, fine, MyNewTool;
    Megfog;
    MoveL Poz1_hengerek_felett, v100, fine, MyNewTool;
    MoveL Poz3_hengerek_felett, v100, fine, MyNewTool;
    MoveL Offs(Poz3_hengerek_felett, 0, 0, -170.8 + felOffset), v100, fine, MyNewTool;
    Elenged;
    MoveL Poz3_hengerek_felett, v100, fine, MyNewTool;

    ! 3. Poz2 alulról (1. henger) ? Poz3 középre
    MoveL Poz2_hengerek_felett, v100, fine, MyNewTool;
    MoveL Offs(Poz2_hengerek_felett, 0, 0, -170.8 + felOffset), v100, fine, MyNewTool;
    Megfog;
    MoveL Poz2_hengerek_felett, v100, fine, MyNewTool;
    MoveL Poz3_hengerek_felett, v100, fine, MyNewTool;
    MoveL Offs(Poz3_hengerek_felett, 0, 0, -125.8 + felOffset), v100, fine, MyNewTool;
    Elenged;
    MoveL Poz3_hengerek_felett, v100, fine, MyNewTool;

    ! 4. Poz1 alulról (3. henger) ? Poz2 alulra
    MoveL Poz1_hengerek_felett, v100, fine, MyNewTool;
    MoveL Offs(Poz1_hengerek_felett, 0, 0, -170.8 + felOffset), v100, fine, MyNewTool;
    Megfog;
    MoveL Poz1_hengerek_felett, v100, fine, MyNewTool;
    MoveL Poz2_hengerek_felett, v100, fine, MyNewTool;
    MoveL Offs(Poz2_hengerek_felett, 0, 0, -170.8 + felOffset), v100, fine, MyNewTool;
    Elenged;
    MoveL Poz2_hengerek_felett, v100, fine, MyNewTool;

    ! 5. Poz3 középrol (1. henger) ? Poz1 alulra
    MoveL Poz3_hengerek_felett, v100, fine, MyNewTool;
    MoveL Offs(Poz3_hengerek_felett, 0, 0, -125.8 + felOffset), v100, fine, MyNewTool;
    Megfog;
    MoveL Poz3_hengerek_felett, v100, fine, MyNewTool;
    MoveL Poz1_hengerek_felett, v100, fine, MyNewTool;
    MoveL Offs(Poz1_hengerek_felett, 0, 0, -170.8 + felOffset), v100, fine, MyNewTool;
    Elenged;
    MoveL Poz1_hengerek_felett, v100, fine, MyNewTool;

    ! 6. Poz3 alulról (2. henger) ? Poz2 középre
    MoveL Poz3_hengerek_felett, v100, fine, MyNewTool;
    MoveL Offs(Poz3_hengerek_felett, 0, 0, -170.8 + felOffset), v100, fine, MyNewTool;
    Megfog;
    MoveL Poz3_hengerek_felett, v100, fine, MyNewTool;
    MoveL Poz2_hengerek_felett, v100, fine, MyNewTool;
    MoveL Offs(Poz2_hengerek_felett, 0, 0, -125.8 + felOffset), v100, fine, MyNewTool;
    Elenged;
    MoveL Poz2_hengerek_felett, v100, fine, MyNewTool;

    ! 7. Poz1 alulról (1. henger) ? Poz2 felülre
    MoveL Poz1_hengerek_felett, v100, fine, MyNewTool;
    MoveL Offs(Poz1_hengerek_felett, 0, 0, -170.8 + felOffset), v100, fine, MyNewTool;
    Megfog;
    MoveL Poz1_hengerek_felett, v100, fine, MyNewTool;
    MoveL Poz2_hengerek_felett, v100, fine, MyNewTool;
    MoveL Offs(Poz2_hengerek_felett, 0, 0, -80.8 + felOffset), v100, fine, MyNewTool;
    Elenged;
    MoveL Poz2_hengerek_felett, v100, fine, MyNewTool;

    MoveL Home, v100, fine, MyNewTool;
ENDPROC

PROC Poz1_Poz3()
    CONST num hMag := 45;
    CONST num felOffset := hMag / 2;

    MoveL Home, v100, fine, MyNewTool\WObj:=wobj0;

    ! 1. Poz1 felülrol (1. henger) ? Poz3 alulra
    MoveL Poz1_hengerek_felett, v100, fine, MyNewTool;
    MoveL Offs(Poz1_hengerek_felett, 0, 0, -80.8 + felOffset), v100, fine, MyNewTool;
    Megfog;
    MoveL Poz1_hengerek_felett, v100, fine, MyNewTool;
    MoveL Poz3_hengerek_felett, v100, fine, MyNewTool;
    MoveL Offs(Poz3_hengerek_felett, 0, 0, -170.8 + felOffset), v100, fine, MyNewTool;
    Elenged;
    MoveL Poz3_hengerek_felett, v100, fine, MyNewTool;

    ! 2. Poz1 középrol (2. henger) ? Poz2 alulra
    MoveL Poz1_hengerek_felett, v100, fine, MyNewTool;
    MoveL Offs(Poz1_hengerek_felett, 0, 0, -125.8 + felOffset), v100, fine, MyNewTool;
    Megfog;
    MoveL Poz1_hengerek_felett, v100, fine, MyNewTool;
    MoveL Poz2_hengerek_felett, v100, fine, MyNewTool;
    MoveL Offs(Poz2_hengerek_felett, 0, 0, -170.8 + felOffset), v100, fine, MyNewTool;
    Elenged;
    MoveL Poz2_hengerek_felett, v100, fine, MyNewTool;

    ! 3. Poz3 alulról (1. henger) ? Poz2 középre
    MoveL Poz3_hengerek_felett, v100, fine, MyNewTool;
    MoveL Offs(Poz3_hengerek_felett, 0, 0, -170.8 + felOffset), v100, fine, MyNewTool;
    Megfog;
    MoveL Poz3_hengerek_felett, v100, fine, MyNewTool;
    MoveL Poz2_hengerek_felett, v100, fine, MyNewTool;
    MoveL Offs(Poz2_hengerek_felett, 0, 0, -125.8 + felOffset), v100, fine, MyNewTool;
    Elenged;
    MoveL Poz2_hengerek_felett, v100, fine, MyNewTool;

    ! 4. Poz1 alulról (3. henger) ? Poz3 alulra
    MoveL Poz1_hengerek_felett, v100, fine, MyNewTool;
    MoveL Offs(Poz1_hengerek_felett, 0, 0, -170.8 + felOffset), v100, fine, MyNewTool;
    Megfog;
    MoveL Poz1_hengerek_felett, v100, fine, MyNewTool;
    MoveL Poz3_hengerek_felett, v100, fine, MyNewTool;
    MoveL Offs(Poz3_hengerek_felett, 0, 0, -170.8 + felOffset), v100, fine, MyNewTool;
    Elenged;
    MoveL Poz3_hengerek_felett, v100, fine, MyNewTool;

    ! 5. Poz2 középrol (1. henger) ? Poz1 alulra
    MoveL Poz2_hengerek_felett, v100, fine, MyNewTool;
    MoveL Offs(Poz2_hengerek_felett, 0, 0, -125.8 + felOffset), v100, fine, MyNewTool;
    Megfog;
    MoveL Poz2_hengerek_felett, v100, fine, MyNewTool;
    MoveL Poz1_hengerek_felett, v100, fine, MyNewTool;
    MoveL Offs(Poz1_hengerek_felett, 0, 0, -170.8 + felOffset), v100, fine, MyNewTool;
    Elenged;
    MoveL Poz1_hengerek_felett, v100, fine, MyNewTool;

    ! 6. Poz2 alulról (2. henger) ? Poz3 középre
    MoveL Poz2_hengerek_felett, v100, fine, MyNewTool;
    MoveL Offs(Poz2_hengerek_felett, 0, 0, -170.8 + felOffset), v100, fine, MyNewTool;
    Megfog;
    MoveL Poz2_hengerek_felett, v100, fine, MyNewTool;
    MoveL Poz3_hengerek_felett, v100, fine, MyNewTool;
    MoveL Offs(Poz3_hengerek_felett, 0, 0, -125.8 + felOffset), v100, fine, MyNewTool;
    Elenged;
    MoveL Poz3_hengerek_felett, v100, fine, MyNewTool;

    ! 7. Poz1 alulról (1. henger) ? Poz3 felülre
    MoveL Poz1_hengerek_felett, v100, fine, MyNewTool;
    MoveL Offs(Poz1_hengerek_felett, 0, 0, -170.8 + felOffset), v100, fine, MyNewTool;
    Megfog;
    MoveL Poz1_hengerek_felett, v100, fine, MyNewTool;
    MoveL Poz3_hengerek_felett, v100, fine, MyNewTool;
    MoveL Offs(Poz3_hengerek_felett, 0, 0, -80.8 + felOffset), v100, fine, MyNewTool;
    Elenged;
    MoveL Poz3_hengerek_felett, v100, fine, MyNewTool;

    MoveL Home, v100, fine, MyNewTool;
ENDPROC

ENDMODULE

--- Backups/IRB140_6_81/RAPID/TASK1/SYSMOD/LINKEDM.sys ---
%%%
  VERSION:1
  LANGUAGE:ENGLISH
%%%

MODULE LINKEDM (SYSMODULE)

! FOLLOWER
!     Name of electronically linked follower axis used by operator at teach pendent.
      PERS string l_f_axis_name{5}       :=  ["",  "", "", "", ""];

!     Name of the mechanical unit for follower axis.
      PERS string l_f_mecunt_n{5}  :=  ["", "", "", "", ""];

!     Linked follower axis number in the mechanical unit (first axis in mech. unit is number 1).
      PERS num l_f_axis_no{5}      :=  [0,          0,   0,  0,  0];

! MASTER
!     Name of the mechanical unit for linked master axis.
      PERS string l_m_mecunt_n{5} :=  ["", "", "", "", ""];

!     Linked master axis number in the mechanical unit (first axis in mech. unit is number 1).
!     See axis number table in documentation for different master mechanical units.
      PERS num l_m_axis_no{5}     :=  [0,  0,  0,  0,  0];

! POSITION OFFSET
!     The increase of the allowed offset position between the master and follower
!     positions, used when starting AUTO mode. As soon as the offset is decreased
!     the old configurated parameter is used.
!     Example: 3 => the configurated value of allowed offset is increased 3 times.
      PERS num offset_ratio{5}       :=  [10,  10,   10,  10,  10];

! SPEED RATIO
!     Speed_ratio used in AUTO and JOG modes [ very_slow   slow    normal    fast]
!     Value 1 = max allowed manual speed.
      CONST num speed_ratio {20}      := [0.01, 0.01, 0.01, 0.01, 0.01,
                                          0.05, 0.05, 0.05, 0.05, 0.05,
                                          0.20, 0.20, 0.20, 0.20, 0.20,
                                          1.00, 1.00, 1.00, 1.00, 1.00];

! STEP SIZE
!     Displacement position used in JOG mode for each activation of positive or
!     negative movement.                  [very_short    short   normal   long]
!     Unit degees or meter.
      CONST num displacement {20}     := [0.001, 0.001, 0.001, 0.001, 0.001,
                                          0.005, 0.005, 0.005, 0.005, 0.005,
                                          0.020, 0.020, 0.020, 0.020, 0.020,
                                          0.100, 0.100, 0.100, 0.100, 0.100];


!-------------------------------------------------------------
 PROC Linked_m ()
      Linked_m_exe ;
 ENDPROC
ENDMODULE

--- Backups/IRB140_6_81/SYSPAR/EIO.cfg ---
EIO:CFG_1.0:6:1::
#
EIO_SIGNAL:

      -Name "DI10_13" -SignalType "DI" -Access "All"

      -Name "DO10_1" -SignalType "DO" -Access "All"

      -Name "DO10_2" -SignalType "DO" -Access "All"

      -Name "DO10_3" -SignalType "DO" -Access "All"

      -Name "DI10_14" -SignalType "DI" -Access "All"
